FUNCTION F_LREAL_TO_STRING : STRING
VAR_INPUT
    Value : LREAL;
    Precision : INT;
END_VAR
VAR
END_VAR

F_LREAL_TO_STRING := LREAL_TO_FMTSTR(in := Value,
                                     iPrecision := Precision,
                                     bRound := TRUE);

END_FUNCTION

(* stored: Version 1.1.0.1, ProductVersion 3.1.4024.3
   POU F_LREAL_TO_STRING: Id {54229989-9fd2-4024-a9b0-09d27c169277}, SpecialFunc None *)
